TYPE Heating_Ctx_Io_Out :
STRUCT
	bPump			: BOOL;
	bBurner			: BOOL;
END_STRUCT
END_TYPE

(* stored: Version 1.1.0.1
   DUT Heating_Ctx_Io_Out: Id {4beac379-8a01-45ac-a9c3-6ceb1387bc53} *)
